FUNCTION_BLOCK "G304M_Code"
TITLE =G304M WITHERING AIR KILN 2
//COPYRIGHT:    (C) 2009  BUHLER AG, CH-9240 UZWIL, SWITZERLAND
//
//PRODUCT:      WinCoS_BIW01_09
//
//TITLE:        WITHERING AIR KILN 2
//                Machine group control
//                Maschinengruppensteuerung
//
//--------------------------------------------------------------------------------
//
//IDENT:        AUTHOR:             DEPT:                              DATE:
//
//P01_FB404.2.0 M.Wedler            AEB41                              27.Apr.2010
//             2nd Release
//P01_FB404.1.0 K.Renz              CSB41                              09.Okt.2009
//             1st Release
//
//--------------------------------------------------------------------------------
//
//PURPOSE:
//
//MANUAL :
//
//RESTRICTIONS:
//
//--------------------------------------------------------------------------------
AUTHOR : KR
FAMILY : USW
VERSION : 9.9


VAR
  Gr : "GCS7_GrpCtrlSub";	//Standard interface to group
  InOutValue1 : DINT ;	//Data for user
  InOutValue2 : DINT ;	//Data for user
  OutWayConflict : BOOL ;	//Data for user
  OutSelectionOk : BOOL ;	//Data for user
  CmdNewValue : BOOL ;	//Data for user
  CmdNewJob : BOOL ;	//Data for user
  OutCodeOK : BOOL ;	//Data for user
  InEndOfJob : BOOL ;	//Data for user
  staWayOk : BOOL ;	//Data for user
  EdgeStartRelease : BOOL ;	//Data for user
  USW8 : BOOL ;	//Data for user
  USW9 : BOOL ;	//Data for user
  USW10 : BOOL ;	//Data for user
  USW11 : BOOL ;	//Data for user
  USW12 : BOOL ;	//Data for user
  USW13 : BOOL ;	//Data for user
  USW14 : BOOL ;	//Data for user
  USW15 : BOOL ;	//Data for user
  A_3245_MXZ11 : "GCS7_E_ValveControl4Pos";	// VLS4Ctrl
  A_3245_MXZ11I1 : "GCS7_E_DigInput";	// DigInpCont
  A_3245_MXZ11I2 : "GCS7_E_DigInput";	// DigInpCont
  A_3246_MXZ11 : "GCS7_E_ValveControl4Pos";	// VLS4Ctrl
  A_3246_MXZ11I1 : "GCS7_E_DigInput";	// DigInpCont
  A_3246_MXZ11I2 : "GCS7_E_DigInput";	// DigInpCont
  A_3245_BZS14 : "GCS7_E_DigInput";	// DigInpCont
  A_3245_BZS15 : "GCS7_E_DigInput";	// DigInpCont
  A_3246_BZS14 : "GCS7_E_DigInput";	// DigInpCont
  A_3246_BZS15 : "GCS7_E_DigInput";	// DigInpCont
END_VAR
VAR_TEMP
  tmpEnable : BOOL ;
  tmpFlag : BOOL ;
  tmpCmdNext : BOOL ;
  tmpLocal : BOOL ;
  tmpAspOk : BOOL ;
  tmpHWStop : BOOL ;
  tmpInstanzDBNo : INT ;
END_VAR
BEGIN
NETWORK
TITLE =



NETWORK
TITLE =Read command from group control
//Parameter
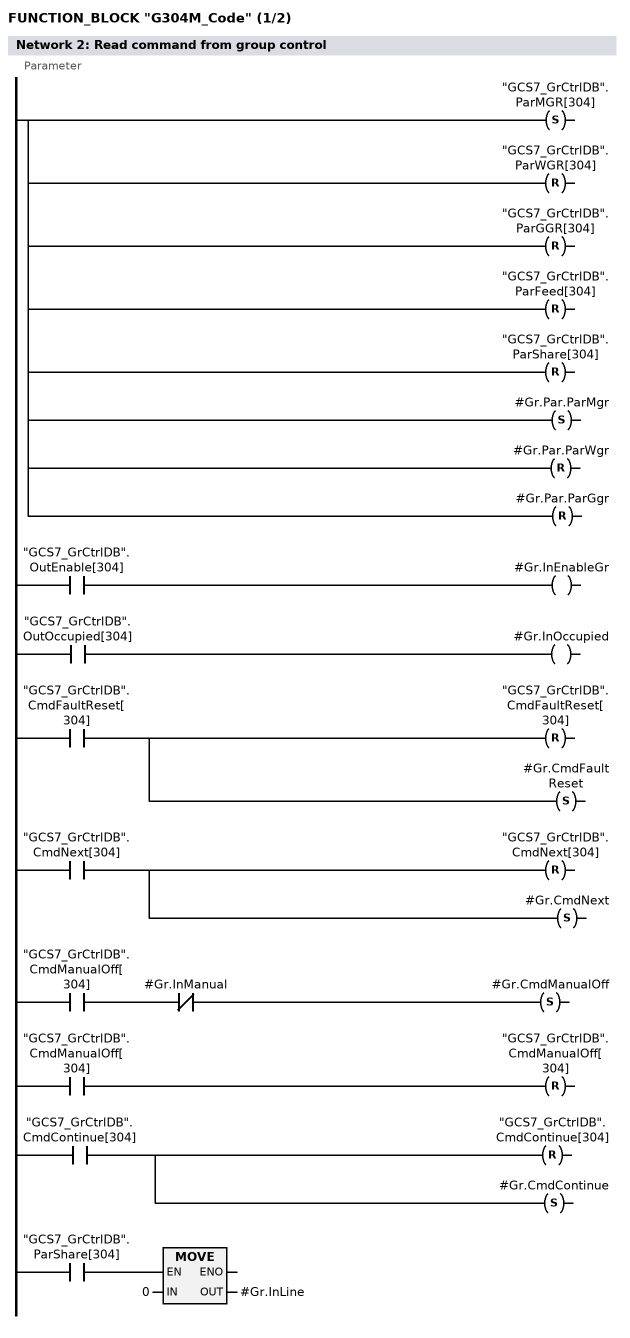
      SET   ;
      S     "GCS7_GrCtrlDB".ParMGR[304];
      R     "GCS7_GrCtrlDB".ParWGR[304];
      R     "GCS7_GrCtrlDB".ParGGR[304];
      R     "GCS7_GrCtrlDB".ParFeed[304];
      R     "GCS7_GrCtrlDB".ParShare[304];
      S     #Gr.Par.ParMgr;
      R     #Gr.Par.ParWgr;
      R     #Gr.Par.ParGgr;
//Command
      U     "GCS7_GrCtrlDB".OutEnable[304];
      =     #Gr.InEnableGr;
      U     "GCS7_GrCtrlDB".OutOccupied[304];
      =     #Gr.InOccupied;
      U     "GCS7_GrCtrlDB".CmdFaultReset[304];
      R     "GCS7_GrCtrlDB".CmdFaultReset[304];
      S     #Gr.CmdFaultReset;
      U     "GCS7_GrCtrlDB".CmdNext[304];
      R     "GCS7_GrCtrlDB".CmdNext[304];
      S     #Gr.CmdNext;

      U     "GCS7_GrCtrlDB".CmdManualOff[304];
      UN    #Gr.InManual;
      S     #Gr.CmdManualOff;
      U     "GCS7_GrCtrlDB".CmdManualOff[304];
      R     "GCS7_GrCtrlDB".CmdManualOff[304];

//      U     "GCS7_GrCtrlDB".CmdManualOff[304]
//      O     "GCS7_GrCtrlDB".OutOccupied[304]
//      R     "GCS7_GrCtrlDB".CmdManualOff[304]
//      S     #Gr.CmdManualOff

      U     "GCS7_GrCtrlDB".CmdContinue[304];
      R     "GCS7_GrCtrlDB".CmdContinue[304];
      S     #Gr.CmdContinue;
//Init Line Number
      U     "GCS7_GrCtrlDB".ParShare[304];
      SPBN  WE00;
      L     0;
      T     #Gr.InLine;
WE00: NOP   0;
NETWORK
TITLE =Call Methode Control
// 1. Handle Interface PCControl
// 2. Prepare mode --> ModePassive,ModeActive,ModeIdling
// 3. Reset global flags of the group
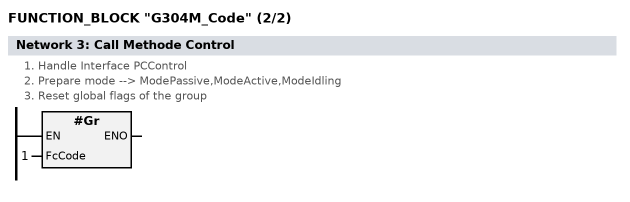
      CALL #Gr (
           FcCode                   := 1);
NETWORK
TITLE =Restart Idling Time

      L     #Gr.Par.ParIdling;
      L     2;
      >=I   ;
      SPB   IdTm;
      T     #Gr.Par.ParIdling;
IdTm: NOP   0;
      U     #A_3245_MXZ11.StNoPosition;
      U     #A_3246_MXZ11.StNoPosition;
      UN    #Gr.InOccupied;
      S     #Gr.CmdRestartIdling;
NETWORK
TITLE =Prepare global flags



NETWORK
TITLE =Set Pattern (Target position)

      U     #Gr.InManual;
      SPB   ILO6;
      L     0; // 0.0%

// Ein-Hordenbetrieb
      U(    ;
      U     "MAL1S033Par".Par.FlagProcess.ProcessEnd; // kilning Process finished
      ON    "MAL1S033Par".Par.FlagProcess.ProcessActive;
      U(    ; //JV290710
      O     "G297M".A_3225_MXZ01MA.Ma.StStopping; //JV290710
      O     "G297M".A_3225_MXZ01MA.Ma.StStopped;
      )     ;
      U(    ;
      O     "G297M".A_3226_MXZ01MA.Ma.StStopping; //JV290710
      O     "G297M".A_3226_MXZ01MA.Ma.StStopped;
      )     ;
      )     ;
      O(    ;
// Zwei-Hordenbetrieb
      U     "MAL1S032Par".Par.FlagProcess.ProcessActive;
      U     "MAL1S033Par".Par.FlagProcess.ProcessActive;
      U     "MAL1S033Par".Par.FlagProcess.Abdarr_Betrieb_Aktiv;
//MW 2010.04.29      U     "G299M".A_3235_MXZ11.StHN
      U     "G299M".A_3236_MXZ11.StHN;
// Klappen im Mischkanal zwischen beden Darren
      U(    ;
//MW 2010.04.29      UN    "G273M".A_3136_MXZ11.StLN
//MW 2010.04.29      UN    "G299M".A_3236_MXZ11.StLN
//MW 2010.04.29      O     "G273M".A_3136_MXZ11.StHN
//MW 2010.04.29      O     "G299M".A_3236_MXZ11.StHN
      UN    "G273M".A_3135_MXZ11.StLN;
      UN    "G299M".A_3235_MXZ11.StLN;
      O     "G273M".A_3135_MXZ11.StHN;
      O     "G299M".A_3235_MXZ11.StHN;
      )     ;
      )     ;
      L     0; //BRT20100826 - hier wurde kein Wert geladen!!!
      SPB   PE;
//    L     "MAL1S033Par".Par.ParIntProcess.PosWitheringAirFlapBasic    // setpoint from recipe
//      L     "MAL1S033Par".Par.ParIntProcess.PosExhaustAirFlapBasic
// Oeffnen der Withering Flaps bei Ueberdruck
//BRT20100826 ====> gibt hier keine Überdruckmessung und bei Öffnen der Klappen entsteht Überdruck am Wärmetasucher!!!
      L     1000;
//      L     "MAL1S033Par".Par.ParIntProcess.PosRecycAirFlapBasic    // setpoint from recipe
      L     "MAL1S033Par".Par.ProcessValue.Value17; // Sollwert Umluftklappen Verbund
      -I    ;
//      U     "MAL1S033Par".Par.FlagProcess.ProcessActive
//      UN    "G302M"._31_R271PE.StFault  // HEAT EXCHANGE PRESSURE < 15mbar
//      SPB   PE
//      L     1000                        // 100.0%
//BRT20100826 <=====
PE:   NOP   0;
//BRT20100827 ====> beide Darren fahren mit vermindeter Drehzahl und 100% Abluft, da Abdarr-Betrieb noch nicht erreicht!!!
      U     "MAL1S032Par".Par.FlagProcess.ProcessActive;
      U     "MAL1S033Par".Par.FlagProcess.ProcessActive;
      UN    "MAL1S032Par".Par.FlagProcess.Abdarr_Betrieb_Aktiv;
      UN    "MAL1S033Par".Par.FlagProcess.Abdarr_Betrieb_Aktiv;
      UN    "MAL1S032Par".Par.FlagProcess.Cooling_Activ;
      UN    "MAL1S033Par".Par.FlagProcess.Cooling_Activ;
      SPBN  Kln1;
      L     1000; // 100% Abluft
Kln1: NOP   0;
//BRT20100827 <=====

//JV260710 =====>   Cooling kiln 2
      U(    ;
      U     "MAL1S033Par".Par.FlagProcess.ProcessActive;
      U     "MAL1S033Par".Par.FlagProcess.Cooling_Activ;
//BRT20100826 ====> im 2 Darren-Betrieb darf auf keinen Fall die Abluft öffnen!!!
      U     "MAL1S032Par".Par.FlagProcess.ProcessActive; // 2 Darren - Betrieb
      UN    "MAL1S033Par".Par.FlagProcess.ProcessEnd;
      UN    M    399.0; //JV090810 Darre 1 kaputt  Hilfsbit zum Kaltblasen Darre 2 über Abluft, nicht zum Kanal
      )     ;
      O(    ;
      UN    "MAL1S033Par".Par.FlagProcess.ProcessActive;
      UN    "MAL1S033Par".Par.FlagProcess.Cooling_Activ;
      U     "MAL1S032Par".Par.FlagProcess.ProcessActive; // 2 Darren - Betrieb
      U     "MAL1S033Par".Par.FlagProcess.ProcessEnd;
      )     ;
      SPBN  Col1;
//      L     1000
//      L     "G273M".A_3135_MXZ11.InPositionMiddle    // Recycling air kiln 1
//      -I
      L     0; //BRT20100825 - Abluft muss zu sein im 2 Darren Kühlschritt
//BRT20100826 <====
Col1: NOP   0; //JV260710 <=====
      U     "G304M".A_3245_MXZ11.InManual;
      SPB   Man1;
      T     #A_3245_MXZ11.InPositionMiddle; // setpoint element
Man1: NOP   0;

      U     "G304M".A_3246_MXZ11.InManual;
      SPB   Man2;
      T     #A_3246_MXZ11.InPositionMiddle; // setpoint element
Man2: NOP   0;
      SPA   En06;
ILO6: NOP   0;
      L     "MAL1S033Par".Par.ParIntProcess.TarPos_ILO_WitheringAir;
      L     10; // convert to 0.1%
      *I    ;
      T     #A_3245_MXZ11.InPositionMiddle; // setpoint element
      T     #A_3246_MXZ11.InPositionMiddle; // setpoint element
En06: NOP   0;

NETWORK
TITLE =Interlocking WayOk



NETWORK
TITLE =Interlocking Autostart

      CLR   ;
      R     #Gr.OutAutostart;
NETWORK
TITLE =Interlocking Enable
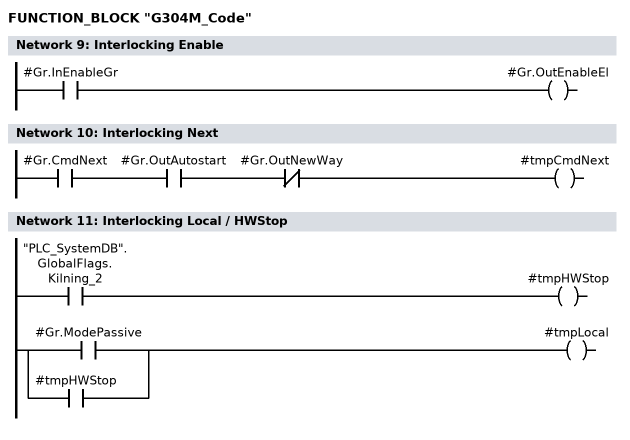

      U     #Gr.InEnableGr;
      =     #Gr.OutEnableEl;

NETWORK
TITLE =Interlocking Next

      U     #Gr.CmdNext;
      U     #Gr.OutAutostart;
      UN    #Gr.OutNewWay;
      =     #tmpCmdNext;

NETWORK
TITLE =Interlocking Local / HWStop

      U     "PLC_SystemDB".GlobalFlags.Kilning_2;
      =     #tmpHWStop;

      U     #Gr.ModePassive;
      O     #tmpHWStop;
      =     #tmpLocal;

NETWORK
TITLE ==A-3245-MXZ11 : LOUVER WITHERING AIR 1

      NOP   0;
//-InLocal---
      U(    ;
      U     #tmpLocal;
      U     #A_3245_BZS14.StTrue;
      O     ;
      U     #Gr.InManual;
      UN    #Gr.InOutAutostartMan;
      )     ;
      =     #A_3245_MXZ11.InLocal;
//
//-Interlocking---
      U     #A_3245_MXZ11.Par.ParManual;
      U     #A_3245_MXZ11.InManual;
      SPB   man1;
      U(    ;
      L     0;
      L     #A_3245_MXZ11.InPositionMiddle; // setpoint element
      ==I   ;
      )     ;
      U(    ;
      U     #Gr.InManual;
      U     #Gr.InOutAutostartMan;
      ON    #Gr.InManual;
      )     ;
      U     #Gr.OutEnableEl;
      =     #A_3245_MXZ11.InLN;

      U(    ;
      L     #A_3245_MXZ11.InPositionMiddle; // setpoint element
      L     0;
      >I    ;
      )     ;
      U(    ;
      L     #A_3245_MXZ11.InPositionMiddle; // setpoint element
      L     1000; // 100,0%
      <I    ;
      )     ;
      U(    ;
      U     #Gr.InManual;
      U     #Gr.InOutAutostartMan;
      ON    #Gr.InManual;
      )     ;
      U     #Gr.OutEnableEl;
      S     #A_3245_MXZ11.CmdMiddle1;

      CLR   ;
      S     #A_3245_MXZ11.CmdMiddle2;

      U(    ;
      UN    #Gr.InOccupied;
      UN    #Gr.InManual;
      )     ;
      O(    ;
      L     #A_3245_MXZ11.InPositionMiddle; // setpoint element
      L     1000; // 100,0%
      >=I   ;
      )     ;
      U(    ;
      U     #Gr.InManual;
      U     #Gr.InOutAutostartMan;
      ON    #Gr.InManual;
      )     ;
      U     #Gr.OutEnableEl;
      S     #A_3245_MXZ11.CmdHN;
man1: NOP   0;
//
//-Read inputs---
//MW      U     "A_3245_MXZ11_I1"
      U     "A_3245_BZS14_I1";
      =     #A_3245_MXZ11.InpLN;
      CLR   ;
      =     #A_3245_MXZ11.InpMiddle1;
//MW      U     "A_3245_MXZ11_I2"
      U     "A_3245_BZS15_I1";
      =     #A_3245_MXZ11.InpHN;
      U     "PLC_SystemDB".GlobalFlags.Kilning_2;
      =     #A_3245_MXZ11.InHWStop;
      U     "PLC_DPInfo".Master[1].SlavesError[101];
      =     #A_3245_MXZ11.InDPFault;
//
//-Set Parameters---
//
//-Call object control---
      CALL #A_3245_MXZ11 ;
//
//-Write outputs---
      U     #A_3245_MXZ11.OutpLN;
      =     "A_3245_MXZ11_O1";
      U     #A_3245_MXZ11.OutpHN;
      =     "A_3245_MXZ11_O2";
NETWORK
TITLE ==A-3245-MXZ11I1 : LOUVER WITHERING AIR 1 CLOSING

      NOP   0;
//-InLocal---
      U     #tmpLocal;
      SET   ;
      =     #A_3245_MXZ11I1.InLocal;
//
//-Monitoring---
      U     #A_3245_MXZ11.OutpLN; // closing
      =     #A_3245_MXZ11I1.InMonTrue;
      CLR   ;
      =     #A_3245_MXZ11I1.InMonFalse;
//
//-PreAlarm---
      CLR   ;
      =     #A_3245_MXZ11I1.InPreAlarmTrue;
      CLR   ;
      =     #A_3245_MXZ11I1.InPreAlarmFalse;
//
//-Additional commands---
//      CLR
//      S     #A_3245_MXZ11I1.CmdRunTimeOutTime
//
//-Read inputs---
      U     "A_3245_MXZ11_I1";
      =     #A_3245_MXZ11I1.InpTrue;
      U     "PLC_SystemDB".GlobalFlags.Kilning_2;
      =     #A_3245_MXZ11I1.InHWStop;
      U     "PLC_DPInfo".Master[1].SlavesError[101];
      =     #A_3245_MXZ11I1.InDPFault;
//
//-Set Parameters---
//
//-Call object control---
      CALL #A_3245_MXZ11I1 ;
//
//-Write outputs---
NETWORK
TITLE ==A-3245-MXZ11I2 : LOUVER WITHERING AIR 1 OPENING

      NOP   0;
//-InLocal---
      U     #tmpLocal;
      SET   ;
      =     #A_3245_MXZ11I2.InLocal;
//
//-Monitoring---
      U     #A_3245_MXZ11.OutpHN; // opening
      =     #A_3245_MXZ11I2.InMonTrue;
      CLR   ;
      =     #A_3245_MXZ11I2.InMonFalse;
//
//-PreAlarm---
      CLR   ;
      =     #A_3245_MXZ11I2.InPreAlarmTrue;
      CLR   ;
      =     #A_3245_MXZ11I2.InPreAlarmFalse;
//
//-Additional commands---
//      CLR
//      S     #A_3245_MXZ11I2.CmdRunTimeOutTime
//
//-Read inputs---
      U     "A_3245_MXZ11_I2";
      =     #A_3245_MXZ11I2.InpTrue;
      U     "PLC_SystemDB".GlobalFlags.Kilning_2;
      =     #A_3245_MXZ11I2.InHWStop;
      U     "PLC_DPInfo".Master[1].SlavesError[101];
      =     #A_3245_MXZ11I2.InDPFault;
//
//-Set Parameters---
//
//-Call object control---
      CALL #A_3245_MXZ11I2 ;
//
//-Write outputs---
NETWORK
TITLE ==A-3246-MXZ11 : LOUVER WITHERING AIR 2

      NOP   0;
//-InLocal---
      U(    ;
      U     #tmpLocal;
      U     #A_3246_BZS14.StTrue;
      O     ;
      U     #Gr.InManual;
      UN    #Gr.InOutAutostartMan;
      )     ;
      =     #A_3246_MXZ11.InLocal;
//
//-Interlocking---
      U     #A_3246_MXZ11.Par.ParManual;
      U     #A_3246_MXZ11.InManual;
      SPB   man2;
      U(    ;
      L     0;
      L     #A_3246_MXZ11.InPositionMiddle; // setpoint element
      ==I   ;
      )     ;
      U(    ;
      U     #Gr.InManual;
      U     #Gr.InOutAutostartMan;
      ON    #Gr.InManual;
      )     ;
      U     #Gr.OutEnableEl;
      =     #A_3246_MXZ11.InLN;

      U(    ;
      L     #A_3246_MXZ11.InPositionMiddle; // setpoint element
      L     0;
      >I    ;
      )     ;
      U(    ;
      L     #A_3246_MXZ11.InPositionMiddle; // setpoint element
      L     1000; // 100,0%
      <I    ;
      )     ;
      U(    ;
      U     #Gr.InManual;
      U     #Gr.InOutAutostartMan;
      ON    #Gr.InManual;
      )     ;
      U     #Gr.OutEnableEl;
      S     #A_3246_MXZ11.CmdMiddle1;

      CLR   ;
      S     #A_3246_MXZ11.CmdMiddle2;

      U(    ;
      UN    #Gr.InOccupied;
      UN    #Gr.InManual;
      )     ;
      O(    ;
      L     #A_3246_MXZ11.InPositionMiddle; // setpoint element
      L     1000; // 100,0%
      >=I   ;
      )     ;
      U(    ;
      U     #Gr.InManual;
      U     #Gr.InOutAutostartMan;
      ON    #Gr.InManual;
      )     ;
      U     #Gr.OutEnableEl;
      S     #A_3246_MXZ11.CmdHN;
      NOP   0;
man2: NOP   0;
//
//-Read inputs---
//MW      U     "A_3246_MXZ11_I1"
      U     "A_3246_BZS14_I1";
      =     #A_3246_MXZ11.InpLN;
      CLR   ;
      =     #A_3246_MXZ11.InpMiddle1;
//MW      U     "A_3246_MXZ11_I2"
      U     "A_3246_BZS15_I1";
      =     #A_3246_MXZ11.InpHN;
      U     "PLC_SystemDB".GlobalFlags.Kilning_2;
      =     #A_3246_MXZ11.InHWStop;
      U     "PLC_DPInfo".Master[1].SlavesError[101];
      =     #A_3246_MXZ11.InDPFault;
//
//-Set Parameters---
//
//-Call object control---
      CALL #A_3246_MXZ11 ;
//
//-Write outputs---
      U     #A_3246_MXZ11.OutpLN;
      =     "A_3246_MXZ11_O1";
      U     #A_3246_MXZ11.OutpHN;
      =     "A_3246_MXZ11_O2";
NETWORK
TITLE ==A-3246-MXZ11I1 : LOUVER WITHERING AIR 2 CLOSING

      NOP   0;
//-InLocal---
      U     #tmpLocal;
      SET   ;
      =     #A_3246_MXZ11I1.InLocal;
//
//-Monitoring---
      U     #A_3246_MXZ11.OutpLN; // closing
      =     #A_3246_MXZ11I1.InMonTrue;
      CLR   ;
      =     #A_3246_MXZ11I1.InMonFalse;
//
//-PreAlarm---
      CLR   ;
      =     #A_3246_MXZ11I1.InPreAlarmTrue;
      CLR   ;
      =     #A_3246_MXZ11I1.InPreAlarmFalse;
//
//-Additional commands---
//      CLR
//      S     #A_3246_MXZ11I1.CmdRunTimeOutTime
//
//-Read inputs---
      U     "A_3246_MXZ11_I1";
      =     #A_3246_MXZ11I1.InpTrue;
      U     "PLC_SystemDB".GlobalFlags.Kilning_2;
      =     #A_3246_MXZ11I1.InHWStop;
      U     "PLC_DPInfo".Master[1].SlavesError[101];
      =     #A_3246_MXZ11I1.InDPFault;
//
//-Set Parameters---
//
//-Call object control---
      CALL #A_3246_MXZ11I1 ;
//
//-Write outputs---
NETWORK
TITLE ==A-3246-MXZ11I2 : LOUVER WITHERING AIR 2 OPENING

      NOP   0;
//-InLocal---
      U     #tmpLocal;
      SET   ;
      =     #A_3246_MXZ11I2.InLocal;
//
//-Monitoring---
      U     #A_3246_MXZ11.OutpHN; // opening
      =     #A_3246_MXZ11I2.InMonTrue;
      CLR   ;
      =     #A_3246_MXZ11I2.InMonFalse;
//
//-PreAlarm---
      CLR   ;
      =     #A_3246_MXZ11I2.InPreAlarmTrue;
      CLR   ;
      =     #A_3246_MXZ11I2.InPreAlarmFalse;
//
//-Additional commands---
//      CLR
//      S     #A_3246_MXZ11I2.CmdRunTimeOutTime
//
//-Read inputs---
      U     "A_3246_MXZ11_I2";
      =     #A_3246_MXZ11I2.InpTrue;
      U     "PLC_SystemDB".GlobalFlags.Kilning_2;
      =     #A_3246_MXZ11I2.InHWStop;
      U     "PLC_DPInfo".Master[1].SlavesError[101];
      =     #A_3246_MXZ11I2.InDPFault;
//
//-Set Parameters---
//
//-Call object control---
      CALL #A_3246_MXZ11I2 ;
//
//-Write outputs---
NETWORK
TITLE ==A-3245-BZS14 : LOUVER WITHERING AIR 1 CLOSED

      NOP   0;
//-InLocal---
      U     #tmpLocal;
      =     #A_3245_BZS14.InLocal;
//
//-Monitoring---
      CLR   ;
      =     #A_3245_BZS14.InMonTrue;
      CLR   ;
      =     #A_3245_BZS14.InMonFalse;
//
//-PreAlarm---
      CLR   ;
      =     #A_3245_BZS14.InPreAlarmTrue;
      CLR   ;
      =     #A_3245_BZS14.InPreAlarmFalse;
//
//-Additional commands---
//      CLR
//      S     #A_3245_BZS14.CmdRunTimeOutTime
//
//-Read inputs---
      U     "A_3245_BZS14_I1";
      =     #A_3245_BZS14.InpTrue;
      U     "PLC_SystemDB".GlobalFlags.Kilning_2;
      =     #A_3245_BZS14.InHWStop;
      U     "PLC_DPInfo".Master[1].SlavesError[101];
      =     #A_3245_BZS14.InDPFault;
//
//-Set Parameters---
//
//-Call object control---
      CALL #A_3245_BZS14 ;
//
//-Write outputs---
NETWORK
TITLE ==A-3245-BZS15 : LOUVER WITHERING AIR 1 OPENED

      NOP   0;
//-InLocal---
      U     #tmpLocal;
      =     #A_3245_BZS15.InLocal;
//
//-Monitoring---
      CLR   ;
      =     #A_3245_BZS15.InMonTrue;
      CLR   ;
      =     #A_3245_BZS15.InMonFalse;
//
//-PreAlarm---
      CLR   ;
      =     #A_3245_BZS15.InPreAlarmTrue;
      CLR   ;
      =     #A_3245_BZS15.InPreAlarmFalse;
//
//-Additional commands---
//      CLR
//      S     #A_3245_BZS15.CmdRunTimeOutTime
//
//-Read inputs---
      U     "A_3245_BZS15_I1";
      =     #A_3245_BZS15.InpTrue;
      U     "PLC_SystemDB".GlobalFlags.Kilning_2;
      =     #A_3245_BZS15.InHWStop;
      U     "PLC_DPInfo".Master[1].SlavesError[101];
      =     #A_3245_BZS15.InDPFault;
//
//-Set Parameters---
//
//-Call object control---
      CALL #A_3245_BZS15 ;
//
//-Write outputs---
NETWORK
TITLE ==A-3246-BZS14 : LOUVER WITHERING AIR 2 CLOSED

      NOP   0;
//-InLocal---
      U     #tmpLocal;
      =     #A_3246_BZS14.InLocal;
//
//-Monitoring---
      CLR   ;
      =     #A_3246_BZS14.InMonTrue;
      CLR   ;
      =     #A_3246_BZS14.InMonFalse;
//
//-PreAlarm---
      CLR   ;
      =     #A_3246_BZS14.InPreAlarmTrue;
      CLR   ;
      =     #A_3246_BZS14.InPreAlarmFalse;
//
//-Additional commands---
//      CLR
//      S     #A_3246_BZS14.CmdRunTimeOutTime
//
//-Read inputs---
      U     "A_3246_BZS14_I1";
      =     #A_3246_BZS14.InpTrue;
      U     "PLC_SystemDB".GlobalFlags.Kilning_2;
      =     #A_3246_BZS14.InHWStop;
      U     "PLC_DPInfo".Master[1].SlavesError[101];
      =     #A_3246_BZS14.InDPFault;
//
//-Set Parameters---
//
//-Call object control---
      CALL #A_3246_BZS14 ;
//
//-Write outputs---
NETWORK
TITLE ==A-3246-BZS15 : LOUVER WITHERING AIR 2 OPENED

      NOP   0;
//-InLocal---
      U     #tmpLocal;
      =     #A_3246_BZS15.InLocal;
//
//-Monitoring---
      CLR   ;
      =     #A_3246_BZS15.InMonTrue;
      CLR   ;
      =     #A_3246_BZS15.InMonFalse;
//
//-PreAlarm---
      CLR   ;
      =     #A_3246_BZS15.InPreAlarmTrue;
      CLR   ;
      =     #A_3246_BZS15.InPreAlarmFalse;
//
//-Additional commands---
//      CLR
//      S     #A_3246_BZS15.CmdRunTimeOutTime
//
//-Read inputs---
      U     "A_3246_BZS15_I1";
      =     #A_3246_BZS15.InpTrue;
      U     "PLC_SystemDB".GlobalFlags.Kilning_2;
      =     #A_3246_BZS15.InHWStop;
      U     "PLC_DPInfo".Master[1].SlavesError[101];
      =     #A_3246_BZS15.InDPFault;
//
//-Set Parameters---
//
//-Call object control---
      CALL #A_3246_BZS15 ;
//
//-Write outputs---
NETWORK
TITLE =Test Fault
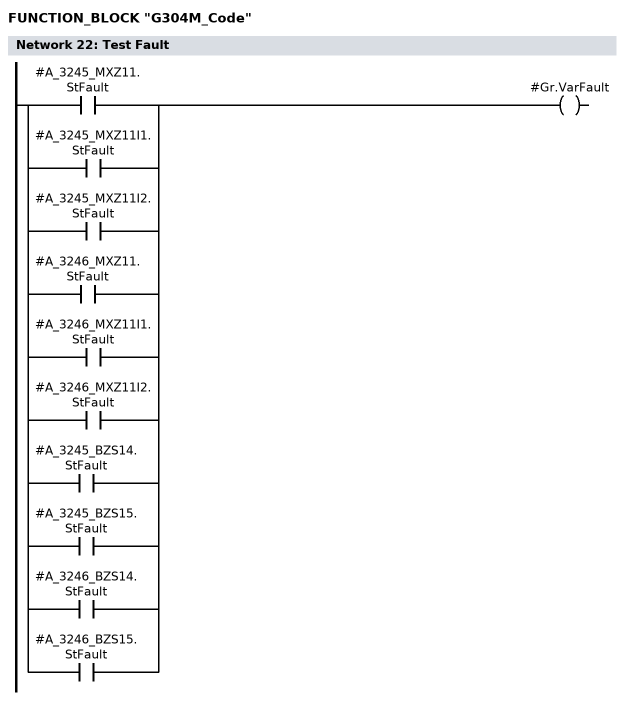

      U     #A_3245_MXZ11.StFault;
      O     #A_3245_MXZ11I1.StFault;
      O     #A_3245_MXZ11I2.StFault;
      O     #A_3246_MXZ11.StFault;
      O     #A_3246_MXZ11I1.StFault;
      O     #A_3246_MXZ11I2.StFault;
      O     #A_3245_BZS14.StFault;
      O     #A_3245_BZS15.StFault;
      O     #A_3246_BZS14.StFault;
      O     #A_3246_BZS15.StFault;
      =     #Gr.VarFault;
NETWORK
TITLE =Test Warning

      CLR   ;
      =     #Gr.OutWarning;
NETWORK
TITLE =Test Stopped
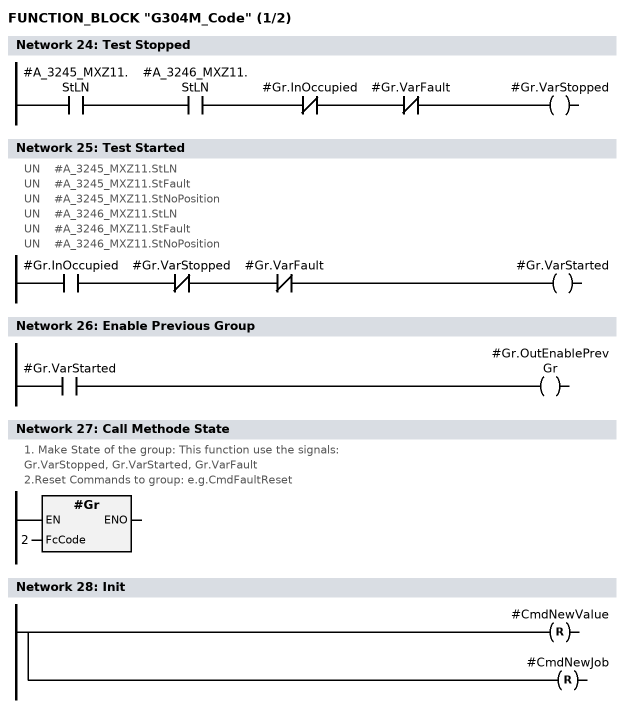

      U     #A_3245_MXZ11.StLN;
      U     #A_3246_MXZ11.StLN;
      UN    #Gr.InOccupied;
      UN    #Gr.VarFault;
      =     #Gr.VarStopped;
NETWORK
TITLE =Test Started
//      UN    #A_3245_MXZ11.StLN
//      UN    #A_3245_MXZ11.StFault
//      UN    #A_3245_MXZ11.StNoPosition
//      UN    #A_3246_MXZ11.StLN
//      UN    #A_3246_MXZ11.StFault
//      UN    #A_3246_MXZ11.StNoPosition
//
      U     #Gr.InOccupied;
      UN    #Gr.VarStopped;
      UN    #Gr.VarFault;
      =     #Gr.VarStarted;
NETWORK
TITLE =Enable Previous Group

      U     #Gr.VarStarted;
      =     #Gr.OutEnablePrevGr;
NETWORK
TITLE =Call Methode State
//1. Make State of the group: This function use the signals:
//        Gr.VarStopped, Gr.VarStarted, Gr.VarFault
//2.Reset Commands to group: e.g.CmdFaultReset
      CALL #Gr (
           FcCode                   := 2);
NETWORK
TITLE =Init

      SET   ;
      R     #CmdNewValue;
      R     #CmdNewJob;
NETWORK
TITLE =Write data to group control
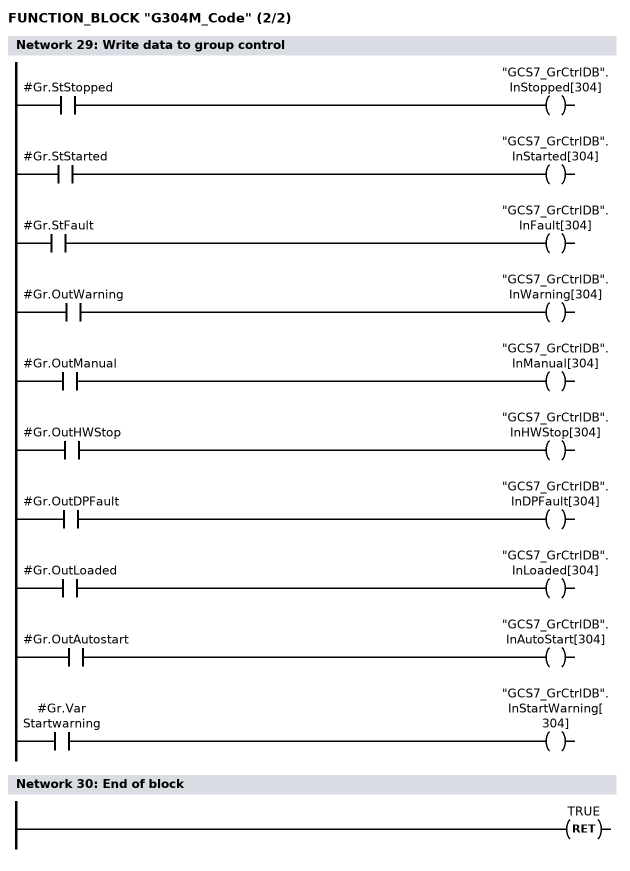

      U     #Gr.StStopped;
      =     "GCS7_GrCtrlDB".InStopped[304];
      U     #Gr.StStarted;
      =     "GCS7_GrCtrlDB".InStarted[304];
      U     #Gr.StFault;
      =     "GCS7_GrCtrlDB".InFault[304];
      U     #Gr.OutWarning;
      =     "GCS7_GrCtrlDB".InWarning[304];
      U     #Gr.OutManual;
      =     "GCS7_GrCtrlDB".InManual[304];
      U     #Gr.OutHWStop;
      =     "GCS7_GrCtrlDB".InHWStop[304];
      U     #Gr.OutDPFault;
      =     "GCS7_GrCtrlDB".InDPFault[304];
      U     #Gr.OutLoaded;
      =     "GCS7_GrCtrlDB".InLoaded[304];
      U     #Gr.OutAutostart;
      =     "GCS7_GrCtrlDB".InAutoStart[304];
      U     #Gr.VarStartwarning;
      =     "GCS7_GrCtrlDB".InStartWarning[304];
NETWORK
TITLE =End of block

      BE    ;

END_FUNCTION_BLOCK

